// TwinCAT 3 PLC project Untitled1
// ProgramVersion: 3.1.4023.0
// libraries:
//   Tc2_Standard, * (Beckhoff Automation GmbH)
//   Tc2_System, * (Beckhoff Automation GmbH)
//   Tc3_Module, * (Beckhoff Automation GmbH)
// project tree:
//   / PlcTask.TcTTO
//   POUs/ MAIN.TcPOU
// real-time tasks:
//   TASK PlcTask: cycle T#50us, priority 20, ADS port 350
// I/O:
//   DEVICE Device 1 (EtherCAT), AmsNetId 134.79.83.3.2.1
//     Term 1 (EK1100) [EK1100 EtherCAT Coupler (2A E-Bus)]
//       Term 2 (EL1004) [EL1004 4Ch. Dig. Input 24V, 3ms]
//       Term 3 (EL2212) [EL2212 2Ch. dig. output with overexcitation (24V DC, 2.5A, 10A Peak)]
//       Term 4 (EL2212) [EL2212 2Ch. dig. output with overexcitation (24V DC, 2.5A, 10A Peak)]
//       Term 5 (EL9011) [EL9011 End Terminal]
// variable links:
//   Untitled1/Untitled1 Instance <-> Device 1 (EtherCAT)/Term 1 (EK1100)/Term 2 (EL1004)
//     PlcTask Inputs/MAIN.close_limit <-> Channel 1/Input
//     PlcTask Inputs/MAIN.open_limit <-> Channel 2/Input
//   Untitled1/Untitled1 Instance <-> Device 1 (EtherCAT)/Term 1 (EK1100)/Term 4 (EL2212)
//     PlcTask Outputs/MAIN.close_pin <-> DOX Control Channel 1/Control/Output
//     PlcTask Outputs/MAIN.open_pin <-> DOX Control Channel 2/Control/Output

CONFIGURATION Untitled1
    RESOURCE PLC ON TwinCAT3
        TASK PlcTask(INTERVAL := T#50us, PRIORITY := 20);
        PROGRAM MAIN WITH PlcTask : MAIN;
    END_RESOURCE
END_CONFIGURATION

// ---- POUs/MAIN.TcPOU
PROGRAM MAIN
VAR
	open_directive		: 	BOOL;
	delay 				:	LINT;
	delay_timer_limit	:	LINT;
	open_pin 	AT%Q* 	: 	BOOL;
	close_pin 	AT%Q* 	:	BOOL;
	
	open_limit 	AT%I*	: 	BOOL;
	close_limit AT%I*	: 	BOOL;
END_VAR


IF NOT open_directive THEN
	IF delay < delay_timer_limit THEN
		delay := delay+ 1;
	END_IF
ELSE
	delay := 0;
END_IF

IF delay >= delay_timer_limit THEN
	close_pin := TRUE;
ELSE
	close_pin := FALSE;
END_IF

open_pin := open_directive;
(*
IF NOT open_limit THEN
	open_pin := open_directive;
ELSE
	open_PIN := FALSE;
END_IF
*)

END_PROGRAM
